FUNCTION_BLOCK StructTests
VAR
	seed       : UDINT;
	pack_none  : PackNone;
	pack_two   : PackTwo;
	pack_four  : PackFour;
	pack_eight : PackEight;
END_VAR

// All four structs share the same fields and the same seed-driven formula.
// b1  = (seed MOD 2 = 0)
// d1  = seed
// b2  = (seed MOD 3 = 0)
// lw1 = LWORD(seed) * LWORD(3)
pack_none.b1  := (seed MOD 2 = 0);
pack_none.d1  := seed;
pack_none.b2  := (seed MOD 3 = 0);
pack_none.lw1 := UDINT_TO_LWORD(seed) * UDINT_TO_LWORD(3);

pack_two.b1  := pack_none.b1;
pack_two.d1  := pack_none.d1;
pack_two.b2  := pack_none.b2;
pack_two.lw1 := pack_none.lw1;

pack_four.b1  := pack_none.b1;
pack_four.d1  := pack_none.d1;
pack_four.b2  := pack_none.b2;
pack_four.lw1 := pack_none.lw1;

pack_eight.b1  := pack_none.b1;
pack_eight.d1  := pack_none.d1;
pack_eight.b2  := pack_none.b2;
pack_eight.lw1 := pack_none.lw1;

END_FUNCTION_BLOCK

(* stored: Version 1.1.0.1, ProductVersion 3.1.4024.13
   POU StructTests: Id {b1c2d3e4-0000-4000-8000-000000000001}, SpecialFunc None *)
